{attribute 'qualified_only'}
VAR_GLOBAL
  
END_VAR

(* stored: Version 1.1.0.1, ProductVersion 3.1.4024.12
   GVL GVL: Id {42b3dea9-343a-46cc-bcac-c35cfbf4405a} *)
